FUNCTION_BLOCK EL1008
VAR
	_io : EL1xx8_Data;
	{attribute addProperty Name "WcState"}
	_wcState : WcStateInputToggle;
	{attribute addProperty Name "Info data"}
	_infoData : InfoDataBase;
END_VAR

PROPERTY IO : REFERENCE TO EL1xx8_Data
GET
IO REF= _io;
END_GET
END_PROPERTY

PROPERTY WcState : REFERENCE TO WcStateInputToggle
GET
WcState REF= _wcState;
END_GET
END_PROPERTY

END_FUNCTION_BLOCK

(* stored: Version 1.1.0.1, ProductVersion 3.1.4024.9
   POU EL1008: Id {c1a3e75e-5875-0559-077e-5b6483ea86af}, SpecialFunc None
   Property IO: Id {a8869efd-7418-0758-2387-716e7a772f60}
   Get Get: Id {a4a89d3c-eca8-066e-0377-cf16af365f2a}
   Property WcState: Id {1f28abc2-75cc-0765-20bf-07696982a777}
   Get Get: Id {7d7ec759-8c94-0de8-1e1b-7b8c1cafb61d} *)
